TYPE ST_FILE_LOGGER_SERVICE :
STRUCT
	doFileFlush:			BOOL;							// Set TRUE when flush is wanted
END_STRUCT
END_TYPE

(* stored: Version 1.1.0.1, ProductVersion 3.1.4026.18
   DUT ST_FILE_LOGGER_SERVICE: Id {28ebcf7a-dc81-0d44-2a9d-f9d58e354ca9} *)
